TYPE ST_Probes_test :
STRUCT
	
	anDistances						: ARRAY[0..9] OF DINT;
	abProbeError					: ARRAY[0..10] OF BOOL;
	bGeneralError					: BOOL;
	anHeightProbe					: ARRAY[0..10] OF DINT;

END_STRUCT
END_TYPE

(* stored: Version 1.1.0.1, ProductVersion 3.1.4024.13
   DUT ST_Probes_test: Id {84e24643-423a-42da-8153-4f00aca97b7f} *)
